INTERFACE ITFGesimuleerdAO

PROPERTY SensorWaarde : int
GET
END_GET
SET
END_SET
END_PROPERTY

END_INTERFACE

(* stored: Version 1.1.0.1
   Itf ITFGesimuleerdAO: Id {226360d6-bab2-4a87-8d8f-b6f553092b9e}
   Property SensorWaarde: Id {b9bb470e-cd44-4777-ac5d-a8bc14a96ec4}
   Get Get: Id {20ae6825-3688-4d4c-b8fc-fb0d9689b3f5}
   Set Set: Id {4a40e179-0da2-40b7-827c-57537548b085} *)
